{attribute addProperty BoxType "EK1100-0000-0018"}
{attribute addProperty Id "Beckhoff_EP4xxxEK1122Beckhoff_EP4xxxEK1122_BB643D5B1920240"}
{attribute addProperty CRC "1035261247"}
{attribute addProperty SizeInBites "1920"}
{attribute addProperty SizeInBytes "240"}
TYPE Beckhoff_EP4xxx_3DB4D53F EXTENDS EK1100_179A0949 :
STRUCT
	{attribute addProperty Name "Beckhoff_EP4xxxEK1122"}
	Beckhoff_EP4xxxEK1122 : Beckhoff_EP4xxxEK1122_BB643D5B;
END_STRUCT
END_TYPE

(* stored: Version 1.2.0.0, ProductVersion 3.1.4024.9
   DUT Beckhoff_EP4xxx_3DB4D53F: Id {03d0b17a-fd71-4c1f-a234-1bd1f9b881eb} *)
